// TwinCAT 3 PLC project Sample
// ProgramVersion: 3.1.4020.2
// libraries:
//   MyLibrary01, * (MyCompany)
//   MyLibrary02, * (MyCompany)
//   Tc2_Standard, * (Beckhoff Automation GmbH)
//   Tc2_System, * (Beckhoff Automation GmbH)
//   Tc3_Module, * (Beckhoff Automation GmbH)
// project tree:
//   / PlcTask.TcTTO
//   POUs/ FB_Foo.TcPOU, MAIN.TcPOU
// (motion and I/O tree: see PLC project library01)
// real-time tasks:
//   TASK PlcTask: cycle T#10ms, priority 20, ADS port 350

CONFIGURATION Sample
    RESOURCE PLC ON TwinCAT3
        TASK PlcTask(INTERVAL := T#10ms, PRIORITY := 20);
        PROGRAM MAIN WITH PlcTask : MAIN;
    END_RESOURCE
END_CONFIGURATION

// ---- POUs/MAIN.TcPOU
PROGRAM MAIN
VAR
	fbFoo1	:	MyNamespace01.FB_Foo;
	fbFoo2	:	MyNamespace02.FB_Foo;
	fbFoo3	:	FB_Foo;
END_VAR

fbFoo1();
fbFoo2();
fbFoo3();

END_PROGRAM

// ---- POUs/FB_Foo.TcPOU
FUNCTION_BLOCK PUBLIC FB_Foo
VAR_INPUT
END_VAR
VAR_OUTPUT
	{attribute 'init_namespace'}
	sNamespace	:	STRING;	
END_VAR
VAR
END_VAR

END_FUNCTION_BLOCK
